FUNCTION Call_Emitter
VAR_INPUT
END_VAR
VAR
END_VAR

instEmitterZufuehrband(PartPresent:= Bauteil_Vorh_Zufuehrb_Ein, 
					   ActorInstanceIndex := 0,
					   ActorInstanceName := 'Part Creation',
					   HMIInterface := hmiMachineSectionInterface,
					   CreatePart=> Bauteil_Erzeugen);
					   
IF NOT Bauteil_Vorh_Zufuehrb_Ein AND 
	currentStateOperatingMode.AutomaticStart.IsActive
THEN
	instEmitterZufuehrband.Create();
END_IF

END_FUNCTION

(* stored: Version 1.1.0.1
   POU Call_Emitter: Id {6e7476dd-b85e-4b73-a561-c0a06f7c7226}, SpecialFunc None *)
